FUNCTION_BLOCK Q_SetAudioVolume_AUS (* Command SetAudioVolume. *)
  (* Standard: ISO 11783-6; Description: Copyright (c) 2022 HR Agrartechnik GmbH This program and the accompanying materials are made available under the terms of the Eclipse Public License 2.0 which is available at https://www.eclipse.org/legal/epl-2.0/ SPDX-License-Identifier: EPL-2.0 see Description Tab *)
  (* Version 1.0, 2025-02-23, Franz Höpfinger, HR Agrartechnik GmbH *)
  PACKAGE isobus::UT::Q;
  (* Documentation:
  Command SetAudioVolume
   This command can be used to control the audio on the VT (volume) ( Part 6 - F.12 )
   param[in] {volume_percent, uint8_t}
   Volume 0 - 100 (%)
   Return Values: 
   int16_t
    - VT_E_NO_ERR (0) - OK
   - VT_E_OVERFLOW (-6) - buffer overflow
   - VT_E_NOACT (-8) - Command not possible in current state
   - VT_E_NO_INSTANCE (-21) - No VT client available
   - VT_E_ISO_INSTANCE_INVALID (-129) - Identifier for instance (connection) invalid
   - VT_E_HANDLE_INVALID (-128) - ErrorCause: invalid Handle
   - VT_E_NOT_ALIVE (-130) - Identifier for instance valid, but VT Dead.
  *)
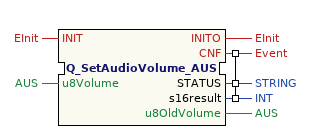
  EVENT_INPUT
    INIT : EInit; (* Service Initialization *)
  END_EVENT
  EVENT_OUTPUT
    INITO : EInit; (* Initialization Confirm *)
    CNF WITH STATUS, s16result; (* Confirmation of Requested Service *)
  END_EVENT
  VAR_OUTPUT
    STATUS : STRING; (* Service Status *)
    s16result : INT; (* retval see description *)
  END_VAR
  SOCKETS
    u8Volume : adapter::types::unidirectional::AUS; (* Volume 0 - 100 (%) *)
  END_SOCKETS
  PLUGS
    u8OldVolume : adapter::types::unidirectional::AUS; (* Old volume 0 - 100 (%) *)
  END_PLUGS
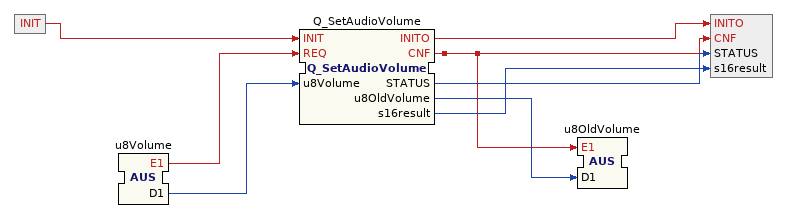
  FBS
    Q_SetAudioVolume : isobus::UT::Q::Q_SetAudioVolume;
  END_FBS
  EVENT_CONNECTIONS
    INIT TO Q_SetAudioVolume.INIT;
    Q_SetAudioVolume.INITO TO INITO;
    Q_SetAudioVolume.CNF TO CNF;
    u8Volume.E1 TO Q_SetAudioVolume.REQ;
    Q_SetAudioVolume.CNF TO u8OldVolume.E1;
  END_CONNECTIONS
  DATA_CONNECTIONS
    Q_SetAudioVolume.STATUS TO STATUS;
    u8Volume.D1 TO Q_SetAudioVolume.u8Volume;
    Q_SetAudioVolume.u8OldVolume TO u8OldVolume.D1;
    Q_SetAudioVolume.s16result TO s16result;
  END_CONNECTIONS
END_FUNCTION_BLOCK
